{attribute 'linkalways'} 
{attribute 'no_explicit_call' := 'This FB is a CLASS and must be accessed using methods or properties'}
{attribute 'enable_dynamic_creation'}
FUNCTION_BLOCK NodePreExecuteEvent EXTENDS Disposable IMPLEMENTS I_NodePreExecuteEvent
VAR
	_target : I_Node;
	_cancelExecute : BOOL;
END_VAR

METHOD PUBLIC Cancel
VAR_INPUT
END_VAR
_cancelExecute := true;
END_METHOD

PROPERTY PUBLIC ExecuteCancelled : BOOL
GET
ExecuteCancelled := _cancelExecute;
END_GET
END_PROPERTY

METHOD FB_init : BOOL
VAR_INPUT
	bInitRetains : BOOL; // if TRUE, the retain variables are initialized (warm start / cold start)
	bInCopyCode : BOOL;  // if TRUE, the instance afterwards gets moved into the copy code (online change)
	Target : I_Node;
END_VAR
_target := Target;
END_METHOD

PROPERTY PUBLIC Target : I_Node
GET
Target := _target;
END_GET
END_PROPERTY

END_FUNCTION_BLOCK

(* stored: Version 1.1.0.1, ProductVersion 3.1.4024.12
   POU NodePreExecuteEvent: Id {c5bd807a-8221-0b85-0548-dc55f13887cb}, SpecialFunc None
   Folder Constructor: Id {40c0e463-c5b7-09ea-2acd-67b8ba9ad94d}
   Method Cancel: Id {6fae4906-bdc2-0d39-2216-10c656cb8723}
   Property ExecuteCancelled: Id {39cb0c5d-437c-08e7-1760-9934ca52051f}
   Get Get: Id {9c7a7a2b-2e42-00c3-3368-e83fffbca03e}
   Method FB_init: Id {c2afc618-e49c-04bc-22e5-eb11cfb4d308}
   Property Target: Id {fb55ddea-3927-004b-322d-079fb1bf38bf}
   Get Get: Id {c9e3ed25-ff10-08d8-2f90-23f32ba015fb} *)
